// TIA Portal V15.1 export
// export: Created 2024-05-17T05:38:24.9670311Z, ExportSetting WithDefaults, DisplayName Totally Integrated Automation Portal, DisplayVersion V15.1 Update 5, DisplayName TIA Portal Openness, DisplayVersion V15.1 Update 5, DisplayName SINAMICS Startdrive Advanced, DisplayVersion V15.1, DisplayName G130, G150, S120, S150, SINAMICS MV, S210, DisplayVersion V15.1, DisplayName G110M, G120, G120C, G120D, G120P, DisplayVersion V15.1, DisplayName STEP 7 Professional, DisplayVersion V15.1 Update 5, DisplayName STEP 7 Safety, DisplayVersion V15.1, DisplayName WinCC Professional, DisplayVersion V15.1 Update 5, DisplayName SIMATIC Visualization Architect, DisplayVersion V15.1
FUNCTION_BLOCK "LGapControlAlarm"   // FB1415, FBD
TITLE = LGapControlAlarm
{ S7_Optimized_Access := 'FALSE' }
AUTHOR : VCC
FAMILY : AlarmHnd
NAME : GapCtrl
VERSION : 1.0
// ================================================================================
// This module is used everywhere one alarm shall be generated when one input 
// photocell becomes false and this photocell signal has to be checked during 
// transfer.
// If the alarm is enable, the photocell may not be deactivated by means of 
// breaking the ray.
// This FB also check the consistency of the photocell. During the period we are 
// sure the photocell must be activated (transfer), the input of the photocell is 
// checked on activity.
// Alarm is disable from HMI, a boolean output is available to inform the upper 
// level and do action in the Alarm summary.
// When the conditions to generate the alarm is disappear, a boolean output is 
// available to inform the upper level that the alarm can be reset.
// The alarm is reset by means of the AlarmResetPB signal.
// ================================================================================
// stored: AutoNumber false, IsIECCheckEnabled false, SetENOAutomatically False, UDAEnableTagReadback false
   VAR_INPUT
      I_GapControl { ExternalAccessible := 'False'; ExternalVisible := 'False'; ExternalWritable := 'False'} : Bool;   // Input signal of the alarm
      I_CheckGapCtrlTrueCond { ExternalAccessible := 'False'; ExternalVisible := 'False'; ExternalWritable := 'False'} : Bool;   // Condition to check gap control photocell on TRUE
      I_CheckGapCtrlFalseCond { ExternalAccessible := 'False'; ExternalVisible := 'False'; ExternalWritable := 'False'} : Bool;   // Condition ot check gap control photocell on FALSE
      I_EnableAlarm { ExternalAccessible := 'False'; ExternalVisible := 'False'; ExternalWritable := 'False'} : Bool := TRUE;   // Enable alarm from upper level
      I_Invisible { ExternalAccessible := 'False'; ExternalVisible := 'False'; ExternalWritable := 'False'} : Bool;   // Invisible
      I_AlarmResetPB { ExternalAccessible := 'False'; ExternalVisible := 'False'; ExternalWritable := 'False'} : Bool;   // Alarm reset pushbutton is activated
   END_VAR
   VAR_OUTPUT
      O_GapControlAlm { ExternalAccessible := 'False'; ExternalVisible := 'False'; ExternalWritable := 'False'} : Bool;   // Gap control Alarm
      O_GapControlTrueAlm { ExternalAccessible := 'False'; ExternalVisible := 'False'; ExternalWritable := 'False'} : Bool;   // Gap control True Alarm
      O_GapControlFalseAlm { ExternalAccessible := 'False'; ExternalVisible := 'False'; ExternalWritable := 'False'} : Bool;   // Gap control False Alarm
      O_AlarmDisabled { ExternalAccessible := 'False'; ExternalVisible := 'False'; ExternalWritable := 'False'} : Bool;   // Alarm disabled from HMI
      O_AlarmABCondition { ExternalAccessible := 'False'; ExternalVisible := 'False'; ExternalWritable := 'False'} : Bool;   // Alarm AB condition
      H_IAnim { ExternalAccessible := 'False'; ExternalVisible := 'False'; ExternalWritable := 'False'} : Word;
   END_VAR
   VAR DB_SPECIFIC
      H_In : Struct   // HMI
         DisableAlarm : Bool;   // Disable alarm from HMI
      END_STRUCT;
      H_Out : Struct   // HMI
         Anim : Word;   // HMI Animation of the object
      END_STRUCT;
      GapControlAlm { ExternalAccessible := 'False'; ExternalVisible := 'False'; ExternalWritable := 'False'} : Bool;   // Gap control Alarm
      GapControlAlmCond { ExternalAccessible := 'False'; ExternalVisible := 'False'; ExternalWritable := 'False'} : Bool;   // Gap control Alarm condition
      PCheckGapTrue { ExternalAccessible := 'False'; ExternalVisible := 'False'; ExternalWritable := 'False'} : Bool;   // Pulse Check detection on True signal
      GapControlTrueMem { ExternalAccessible := 'False'; ExternalVisible := 'False'; ExternalWritable := 'False'} : Bool;   // Memory Gap control on True signal
      GapControlTrueAlm { ExternalAccessible := 'False'; ExternalVisible := 'False'; ExternalWritable := 'False'} : Bool;   // Gap control alarm on True
      GapControlTrueAlmCond { ExternalAccessible := 'False'; ExternalVisible := 'False'; ExternalWritable := 'False'} : Bool;   // Alarm condition of Gap Control True Alarm
      PCheckGapfalse { ExternalAccessible := 'False'; ExternalVisible := 'False'; ExternalWritable := 'False'} : Bool;   // Pulse Check detection on False signal
      GapControlFalseMem { ExternalAccessible := 'False'; ExternalVisible := 'False'; ExternalWritable := 'False'} : Bool;   // Memory Gap control on False signal
      GapControlFalseAlm { ExternalAccessible := 'False'; ExternalVisible := 'False'; ExternalWritable := 'False'} : Bool;   // Gap control alarm on False
      GapControlFalseAlmCond { ExternalAccessible := 'False'; ExternalVisible := 'False'; ExternalWritable := 'False'} : Bool;   // Alarm condition of Gap Control False Alarm
   END_VAR
   VAR_TEMP   // added for the SCL form of the ladder/FBD networks
      _w1 : Bool;
   END_VAR
BEGIN

REGION Network 1: **** 2.2 - Alarms - Alarms Generation **** Condition of the Gap control alarm for the Normal CLOSED input
   // Condition of the Gap control alarm for the Normal CLOSED input
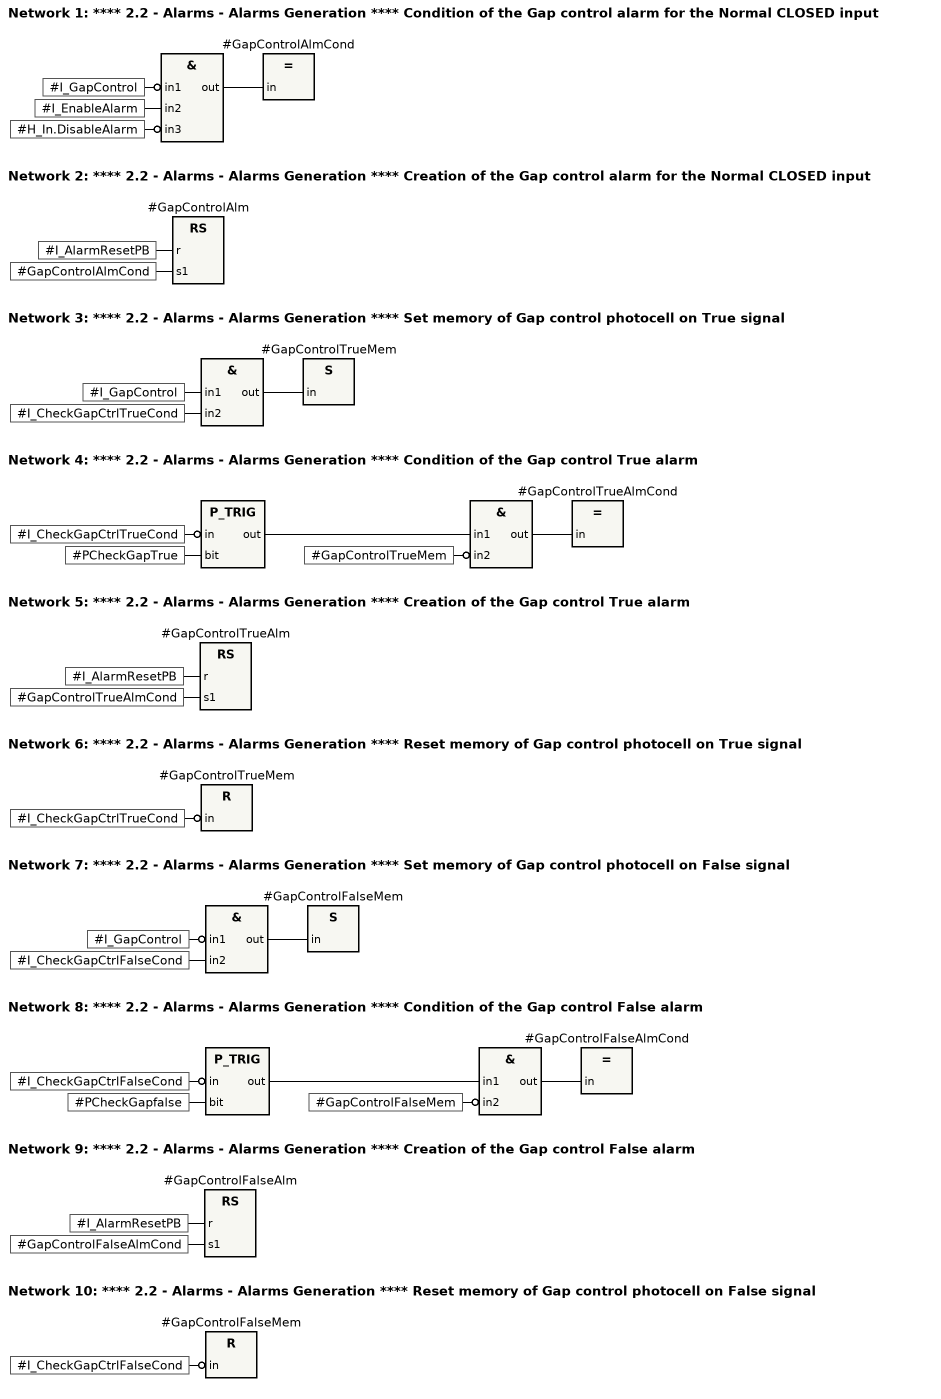
   #GapControlAlmCond := NOT #I_GapControl AND #I_EnableAlarm AND NOT #H_In.DisableAlarm;
END_REGION

REGION Network 2: **** 2.2 - Alarms - Alarms Generation **** Creation of the Gap control alarm for the Normal CLOSED input
   // Creation of the Gap control alarm for the Normal CLOSED input
   IF #I_AlarmResetPB THEN
       #GapControlAlm := FALSE;   // RS flip-flop
   END_IF;
   IF #GapControlAlmCond THEN #GapControlAlm := TRUE; END_IF;
END_REGION

REGION Network 3: **** 2.2 - Alarms - Alarms Generation **** Set memory of Gap control photocell on True signal
   // Set memory of Gap control photocell on True signal
   IF #I_GapControl AND #I_CheckGapCtrlTrueCond THEN #GapControlTrueMem := TRUE; END_IF;
END_REGION

REGION Network 4: **** 2.2 - Alarms - Alarms Generation **** Condition of the Gap control True alarm
   // Condition of the Gap control True alarm
   #_w1 := NOT #I_CheckGapCtrlTrueCond AND NOT #PCheckGapTrue;   // rising edge
   #PCheckGapTrue := NOT #I_CheckGapCtrlTrueCond;
   #GapControlTrueAlmCond := #_w1 AND NOT #GapControlTrueMem;
END_REGION

REGION Network 5: **** 2.2 - Alarms - Alarms Generation **** Creation of the Gap control True alarm
   // Creation of the Gap control True alarm
   IF #I_AlarmResetPB THEN
       #GapControlTrueAlm := FALSE;   // RS flip-flop
   END_IF;
   IF #GapControlTrueAlmCond THEN #GapControlTrueAlm := TRUE; END_IF;
END_REGION

REGION Network 6: **** 2.2 - Alarms - Alarms Generation **** Reset memory of Gap control photocell on True signal
   // Reset memory of Gap control photocell on True signal
   IF NOT #I_CheckGapCtrlTrueCond THEN #GapControlTrueMem := FALSE; END_IF;
END_REGION

REGION Network 7: **** 2.2 - Alarms - Alarms Generation **** Set memory of Gap control photocell on False signal
   // Set memory of Gap control photocell on False signal
   IF NOT #I_GapControl AND #I_CheckGapCtrlFalseCond THEN #GapControlFalseMem := TRUE; END_IF;
END_REGION

REGION Network 8: **** 2.2 - Alarms - Alarms Generation **** Condition of the Gap control False alarm
   // Condition of the Gap control False alarm
   #_w1 := NOT #I_CheckGapCtrlFalseCond AND NOT #PCheckGapfalse;   // rising edge
   #PCheckGapfalse := NOT #I_CheckGapCtrlFalseCond;
   #GapControlFalseAlmCond := #_w1 AND NOT #GapControlFalseMem;
END_REGION

REGION Network 9: **** 2.2 - Alarms - Alarms Generation **** Creation of the Gap control False alarm
   // Creation of the Gap control False alarm
   IF #I_AlarmResetPB THEN
       #GapControlFalseAlm := FALSE;   // RS flip-flop
   END_IF;
   IF #GapControlFalseAlmCond THEN #GapControlFalseAlm := TRUE; END_IF;
END_REGION

REGION Network 10: **** 2.2 - Alarms - Alarms Generation **** Reset memory of Gap control photocell on False signal
   // Reset memory of Gap control photocell on False signal
   IF NOT #I_CheckGapCtrlFalseCond THEN #GapControlFalseMem := FALSE; END_IF;
END_REGION

REGION Network 11: **** 4.6 - Mashine Status - Indications **** Icon Animation
   // Icon Animation
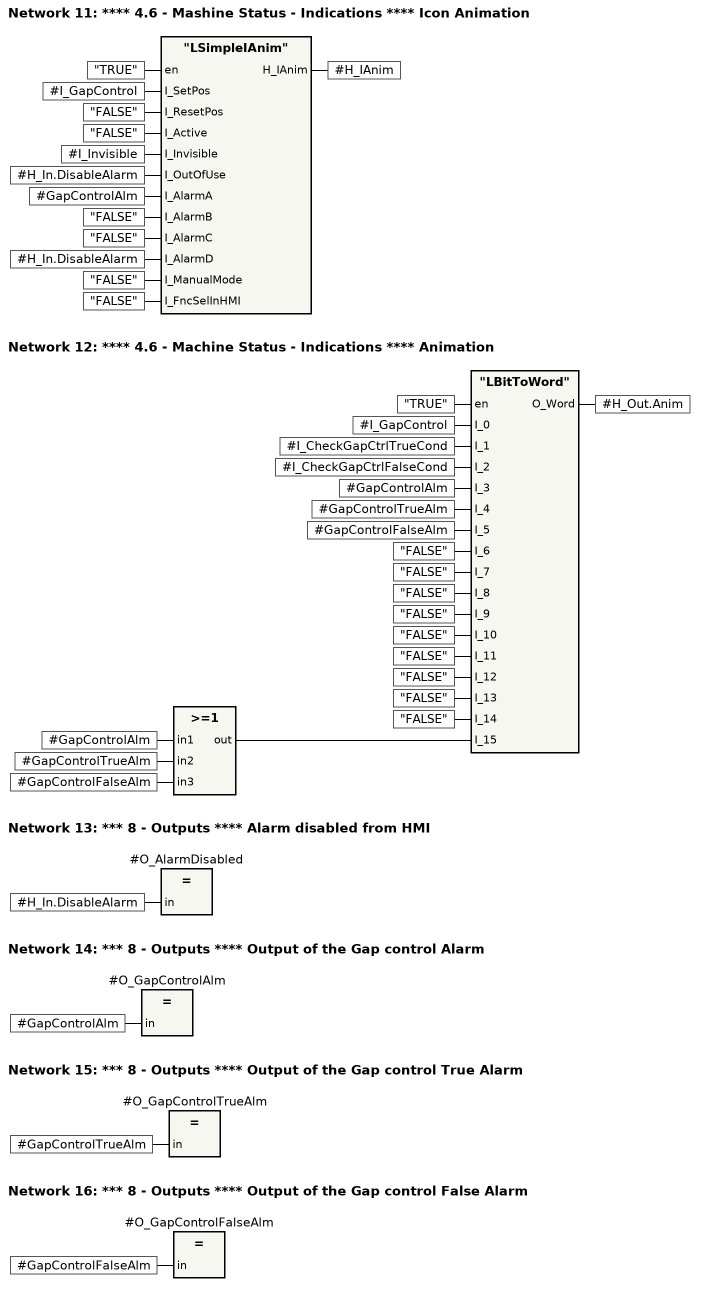
   IF "TRUE" THEN
       "LSimpleIAnim"(I_SetPos := #I_GapControl,
                      I_ResetPos := "FALSE",
                      I_Active := "FALSE",
                      I_Invisible := #I_Invisible,
                      I_OutOfUse := #H_In.DisableAlarm,
                      I_AlarmA := #GapControlAlm,
                      I_AlarmB := "FALSE",
                      I_AlarmC := "FALSE",
                      I_AlarmD := #H_In.DisableAlarm,
                      I_ManualMode := "FALSE",
                      I_FncSelInHMI := "FALSE",
                      H_IAnim => #H_IAnim);
   END_IF;
END_REGION

REGION Network 12: **** 4.6 - Machine Status - Indications **** Animation
   // Animation
   IF "TRUE" THEN
       "LBitToWord"(I_0 := #I_GapControl,
                    I_1 := #I_CheckGapCtrlTrueCond,
                    I_2 := #I_CheckGapCtrlFalseCond,
                    I_3 := #GapControlAlm,
                    I_4 := #GapControlTrueAlm,
                    I_5 := #GapControlFalseAlm,
                    I_6 := "FALSE",
                    I_7 := "FALSE",
                    I_8 := "FALSE",
                    I_9 := "FALSE",
                    I_10 := "FALSE",
                    I_11 := "FALSE",
                    I_12 := "FALSE",
                    I_13 := "FALSE",
                    I_14 := "FALSE",
                    I_15 := #GapControlAlm OR #GapControlTrueAlm OR #GapControlFalseAlm,
                    O_Word => #H_Out.Anim);
   END_IF;
END_REGION

REGION Network 13: *** 8 - Outputs **** Alarm disabled from HMI
   // Alarm disabled from HMI
   #O_AlarmDisabled := #H_In.DisableAlarm;
END_REGION

REGION Network 14: *** 8 - Outputs **** Output of the Gap control Alarm
   // Output of the Gap control Alarm
   #O_GapControlAlm := #GapControlAlm;
END_REGION

REGION Network 15: *** 8 - Outputs **** Output of the Gap control True Alarm
   // Output of the Gap control True Alarm
   #O_GapControlTrueAlm := #GapControlTrueAlm;
END_REGION

REGION Network 16: *** 8 - Outputs **** Output of the Gap control False Alarm
   // Output of the Gap control False Alarm
   #O_GapControlFalseAlm := #GapControlFalseAlm;
END_REGION

REGION Network 17: **** 8 - Outputs **** Alarm resetable
   // Alarm resetable
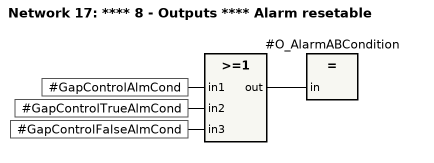
   #O_AlarmABCondition := #GapControlAlmCond OR #GapControlTrueAlmCond OR #GapControlFalseAlmCond;
END_REGION
END_FUNCTION_BLOCK
